TYPE ST_MOVER_OFFSETS :
STRUCT
  // static position offsets in stations
  PositionOffset      : ARRAY[1..MAX_STATION] OF T_NEST_OFFSET; // added to PosStop[] in XtsStation
END_STRUCT
END_TYPE

(* stored: Version 1.1.0.1, ProductVersion 3.1.4026.18
   DUT ST_MOVER_OFFSETS: Id {ce31ad99-7cbc-4102-a4b9-a6a9b8668a17} *)
